(* IEC 61131-3 sources: SamplePLCprogramming/bbi_trail, 4 files *)

(* ---- Types.typ ---- *)
TYPE
	trail_buffer_entry_typ : 	STRUCT
		dat : DATE_AND_TIME;
		ID : UDINT;
		new1 : REAL; (*neuer Prozesswert Real*)
		par1 : UDINT;
		par2 : UDINT;
		string1 : STRING[254];
	END_STRUCT;
	trail_buffer_typ : 	STRUCT
		firstPushed : UINT;
		nextPush : UINT;
		value : ARRAY[0..TRAIL_ENTRIES]OF trail_buffer_entry_typ;
	END_STRUCT;
	eventRecordHeader_typ : 	STRUCT
		deviceident : UDINT; (*Anlagen Id, Batchident*)
		maxBufCount : UDINT; (*Maxiamlanzahl der Events im buffer (statistik)*)
		maxBufSize : UDINT; (*Maximale Datengröße der dateiaktion(statistik)*)
		records : UDINT; (*anzahl der geschriebenen events*)
		crcHeader : UDINT; (*prüfsumme header*)
	END_STRUCT;
END_TYPE

(* ---- bbi_trail.fun ---- *)
FUNCTION_BLOCK fMakeEventData
	VAR_INPUT
		pATbuf : UDINT;
		time : DATE_AND_TIME;
	END_VAR
	VAR_OUTPUT
		data : ARRAY[0..1023] OF USINT; (*könnte aus sicht der aufrufenden instanz auch dataLen heißen*)
		offset : UDINT;
	END_VAR
	VAR
		payloadCountPosition : UDINT;
		CRC : REFERENCE TO UDINT;
		aUDINT : REFERENCE TO UDINT;
		aReal : REFERENCE TO REAL;
		aCRLF : REFERENCE TO ARRAY[0..3] OF USINT;
		i : UINT;
		ebuf : REFERENCE TO trail_buffer_typ;
		indexBuf : UINT;
		e : trail_buffer_entry_typ;
		toMuchData : BOOL;
		eventsToPop : UINT;
	END_VAR
END_FUNCTION_BLOCK

FUNCTION addEvent : UINT (*an cal.isAT hängen*)
	VAR_INPUT
		enable : BOOL;
		pBuf : UDINT;
		event : trail_buffer_entry_typ;
	END_VAR
	VAR
		count : UINT;
		buf : REFERENCE TO trail_buffer_typ;
		e : trail_buffer_entry_typ;
	END_VAR
END_FUNCTION

(* ---- bbi_trail.st ---- *)
FUNCTION addEvent

	(*
		Design einer array queue mit eventstrukturen
		buf.nextPush ist nächster gültiger index für nächstes element, nächsten push dort anhängen
		buf.firstPushed ist zuerst hinzugefügtes element = ältestes, pop dort entnehmen
	*)

	buf ACCESS pBuf;
	e:=event;
	IF NOT enable THEN
		addEvent:=ERR_FUB_ENABLE_FALSE;
	ELSIF pBuf = 0 THEN
		addEvent:=90;		//nullpointer
	ELSE
		IF (buf.firstPushed = buf.nextPush) THEN
			count:=0;
		ELSIF buf.firstPushed > buf.nextPush THEN
			count := TRAIL_ENTRIES - buf.firstPushed + 1 + buf.nextPush;
		ELSE
			count := buf.nextPush - buf.firstPushed;
		END_IF;
		IF count = TRAIL_ENTRIES THEN
			addEvent:=91;		//puffer voll, keine neuen entragungen möglich, ein eintrag muss frei bleiben um leere queue von komplett voller zu unterscheiden
		ELSE
			IF count + 1 = TRAIL_ENTRIES THEN //nur noch ein eintrag (eigentlich zwei) im puffer vorhanden
				e.ID:=18;		//letzter möglicher eintrag, eventuell weitere Events verloren!!!
			END_IF;
			buf.value[buf.nextPush]:=e;
			buf.nextPush := (buf.nextPush + 1)  MOD TRAIL_ENTRIES_COUNT;
			addEvent:=ERR_OK;
		END_IF;
	END_IF;
END_FUNCTION

FUNCTION_BLOCK fMakeEventData //pop für alle werte im puffer
	//start parsing buffer to additional events data in output buffer...
	ebuf ACCESS pATbuf;
	IF (ebuf.firstPushed = ebuf.nextPush) THEN
		eventsToPop:=0;
	ELSIF ebuf.firstPushed > ebuf.nextPush THEN
		eventsToPop := TRAIL_ENTRIES - ebuf.firstPushed + 1 + ebuf.nextPush;
	ELSE
		eventsToPop := ebuf.nextPush - ebuf.firstPushed;
	END_IF;

	IF eventsToPop > 0 THEN //falls einträge vorhanden
		//alle puffereinträge abarbeiten
		indexBuf:=ebuf.firstPushed;
		offset:=0;
		FOR i:=0 TO eventsToPop - 1 BY 1 DO
			//start delimeter erzeugen
			aCRLF ACCESS ADR(data)+offset;
			aCRLF[0]:=DATA_LINE_STARTCHAR5;
			aCRLF[1]:=DATA_LINE_STARTCHAR5;
			aCRLF[2]:=DATA_LINE_STARTCHAR5;
			aCRLF[3]:=DATA_LINE_STARTCHAR5;
			offset:=offset + 4;

			e:=ebuf.value[indexBuf]; //abbild des aktuellen eintrags in e anlegen
			//zeitstempel
			aUDINT ACCESS ADR(data)+offset;
			aUDINT:=DT_TO_UDINT(e.dat); //für alle typen zeit übernehmen
			offset:=offset + 4;
			//für alle typen id schreiben
			aUDINT ACCESS ADR(data)+offset;
			aUDINT:=e.ID;
			offset:=offset + 4;
			payloadCountPosition:=offset; //position des registers der payloadlänge sichern
			offset:=offset + 4;

			CASE e.ID OF
				14,//Reboot
				18,//puffer überlauf (task-übergabe)
				19://puffer überlauf (datei schreiben)
					//keine payload
					1,//login succesfull
					2,//failed
					3,//logout
					5,//PW changed
					6,//reason critical login
					26,//reason cO faceplate
					36,//reason cI fceplate
					37,//reason Cl page
					10,//AT-Start
					70,//Sequenz fordert eingabe an
					75,//Inokulation markiert
				11://AT Stop,
					//par 1			par2		string1
					aUDINT ACCESS ADR(data)+offset;
					aUDINT:=e.par1;
					offset:=offset + 4;

					aUDINT ACCESS ADR(data)+offset;
					aUDINT:=e.par2;
					offset:=offset + 4;

					brsmemcpy(ADR(data)+offset,ADR(e.string1),brsstrlen(ADR(e.string1))+1); //string1;
					offset:=offset + brsstrlen(ADR(e.string1))+1;
					//		aUDINT ACCESS ADR(data)+payloadCountPosition; //länge der payload sichern
					//		aUDINT := offset - payloadCountPosition - 4; //exklusive payload count
					20,//Ausgang geändert
					30,//sollwert aus faceplate ausgänge
				31,34://sollwert aus reglerseite, aus faceplate eingänge

					//par 1			new
					aUDINT ACCESS ADR(data)+offset;
					aUDINT:=e.par1;
					offset:=offset + 4;

					aReal ACCESS ADR(data)+offset;
					aReal:=e.new1;
					offset:=offset + 4;

					22,//lockOff change
					23,//lockman change
					33,//enable regler aus reglerseite
					32,//enable regler aus ausgangsfaceplate
					35,//enable aus eingangsfaceplate
					71,// sequenzdialog OK
					72,// sequenzdialog abbruch
					73,// sequenzdialog timeout
					74,// sequenzdialog minimiert
					40,//profil start/stop
					100,101,102,//alarmsystem
					110,111,112,
					120,121,122,
					130,131,132,
					140,141,142,
					150,151,152,
				160,161,162:
					//par 1			par2
					aUDINT ACCESS ADR(data)+offset;
					aUDINT:=e.par1;
					offset:=offset + 4;

					aUDINT ACCESS ADR(data)+offset;
					aUDINT:=e.par2;
					offset:=offset + 4;
					50,//sequenz manuell gestartet
					51,//sequenz manuell zum herunterfahren aufgefordert
					52,//sequenz zum harten abbruch gezwungen
					55,//sequenz meldet start des herunterfahrens
					56,//hilfs sequenz meldet automatischen start des herunterfahrens nach beenden der muttersequenz
					57,//sequenz meldet erfolg des herunterfahrens
				41://profil ende nach selbstständigem durchlauf
					//par 1
					aUDINT ACCESS ADR(data)+offset;
					aUDINT:=e.par1;
					offset:=offset + 4;
					60,//globaler par geändert vor start der sequenz
				61://globaler par geändert bei laufender sequenz
					//par 1			par2	new 1	string1
					aUDINT ACCESS ADR(data)+offset;
					aUDINT:=e.par1;
					offset:=offset + 4;

					aUDINT ACCESS ADR(data)+offset;
					aUDINT:=e.par2;
					offset:=offset + 4;

					aReal ACCESS ADR(data)+offset;
					aReal:=e.new1;
					offset:=offset + 4;

					brsmemcpy(ADR(data)+offset,ADR(e.string1),brsstrlen(ADR(e.string1))+1); //string1;
					offset:=offset + brsstrlen(ADR(e.string1))+1;
				ELSE //unhandled ID forced to ID 12
					aUDINT ACCESS ADR(data)+offset;
					aUDINT:=e.ID; //unbekannte ID auf par 1 schreiben
					offset:=offset + 4;
					aUDINT ACCESS ADR(data)+offset - 12 ;	//zurückgehen zu e.ID und auf 12 setzen
					aUDINT:=12;
			END_CASE;
			aUDINT ACCESS ADR(data)+payloadCountPosition; //länge der payload sichern
			aUDINT := offset - payloadCountPosition - 4; //exklusive payload count
			//CRC anhängen
			CRC ACCESS ADR(data) + offset;
			CRC:=CRC32(offset - payloadCountPosition + 8,ADR(data) + payloadCountPosition - 8,BATCH_GENERATOR);
			offset:=offset + 4;
			//für jedes event einen  end delimiter erzeugen
			//gleicher end delim wie trenddata, damit offset korrektur kompatibel bleibt
			aCRLF ACCESS ADR(data)+offset;
			aCRLF[0]:=DATA_LINE_ENDCHAR;
			aCRLF[1]:=DATA_LINE_ENDCHAR;
			aCRLF[2]:=13;
			aCRLF[3]:=10;
			offset:=offset + 4;
			//mit jedem  abgearbeitetn eintrag prüfen ob offset + 60 > MAXTRENDDATASIZE,
			toMuchData:=0;
			IF offset + 70 > 1023 THEN //wenigstens platz für einen weiteren eintrag muss noch da sein
				toMuchData:=1;
				i:=eventsToPop;//abort loop
			END_IF;

			//mit einem index für trail buffeer durch die enträge  gehen
			IF indexBuf+1 > TRAIL_ENTRIES THEN
				indexBuf:=0;
			ELSE
				indexBuf:=indexBuf+1;
			END_IF;
		END_FOR;
		IF toMuchData THEN//falls zu viele daten, nur ein event mit ID 19 anlegn
			offset:=0;
			//start delimeter erzeugen
			aCRLF ACCESS ADR(data);
			aCRLF[0]:=DATA_LINE_STARTCHAR5;
			aCRLF[1]:=DATA_LINE_STARTCHAR5;
			aCRLF[2]:=DATA_LINE_STARTCHAR5;
			aCRLF[3]:=DATA_LINE_STARTCHAR5;
			offset:=offset + 4;
			//zeitstempel
			aUDINT ACCESS ADR(data)+offset;
			aUDINT:=DT_TO_UDINT(time); //zeit dieses fehlers übernehmen
			offset:=offset + 4;
			aUDINT ACCESS ADR(data)+offset;
			aUDINT:=19;
			offset:=offset + 4;
			payloadCountPosition:=offset; //position des registers der payloadlänge sichern
			aUDINT ACCESS ADR(data)+offset;
			aUDINT:=0; //für diese event ist payload 0
			offset:=offset + 4;
			//CRC anhängen
			CRC ACCESS ADR(data) + offset;
			CRC:=CRC32(offset - payloadCountPosition + 8,ADR(data) + payloadCountPosition - 8,BATCH_GENERATOR);
			offset:=offset + 4;
			aCRLF ACCESS ADR(data)+offset;
			aCRLF[0]:=DATA_LINE_ENDCHAR;
			aCRLF[1]:=DATA_LINE_ENDCHAR;
			aCRLF[2]:=13;
			aCRLF[3]:=10;
			offset:=offset + 4;
		END_IF;
		ebuf.firstPushed := (ebuf.firstPushed + eventsToPop) MOD (TRAIL_ENTRIES + 1); //puffer um alle gepoppten events bereinigen
	END_IF;

END_FUNCTION_BLOCK

(* ---- Constants.var ---- *)
VAR CONSTANT
	TRAIL_ENTRIES : UINT := 29; (*puffergröße für audittrail events*)
	TRAIL_ENTRIES_COUNT : UINT := TRAIL_ENTRIES + 1; (*maximalanzahl der Enträge = null zeiger*)
END_VAR
